FUNCTION_BLOCK FB_RateFromEPICS

(*
enum MPSBeamRates {
    MPSRateInvalid            =  0,
    MPSRate0Hz                =  1,
    /* Previously used 2 and 3 for single shot and burst */
    MPSRate1Hz                =  4,
    MPSRate10Hz               =  5,
    MPSRate30Hz               =  6,
    MPSRate60Hz               =  7,
    MPSRate120Hz              =  8,
    MPSRateUnknown            =  9,
    MPSRateSingleShot         = 10,
    MPSRateBurstMode          = 11,
    MPSRateBurstModeNotActive = 12,
    MPSNumberOfBeamRates      = 13,
    MPSRateBurstInvalid       = 14
}
*)

VAR_IN_OUT
    BP : ST_BeamParams;
    fbBYKIK_Rate : FB_LREALFromEPICS;
    FFO : FB_HardwareFFOutput;
END_VAR
VAR_OUTPUT
    xError : BOOL;
END_VAR
VAR


    eMPSRate : E_MPSBeamRates;

    ffRateReadBack : FB_FastFault := (
        i_DevName := 'Arbiter',
        i_Desc := 'Issue with rate readback from Accelerator. Gateway or EPICS connection. Must be fixed.',
        i_TypeCode := 16#203,
        i_xAutoReset:=True);
END_VAR
VAR CONSTANT
    cFailSafeRate : UDINT := 1000001;
END_VAR

fbBYKIK_Rate();

IF fbBYKIK_Rate.bValid THEN
    eMPSRate := LREAL_TO_UINT(fbBYKIK_Rate.fValue);
ELSE
    eMPSRate := E_MPSBeamRates.MPSRateInvalid;
END_IF

CASE eMPSRate OF
    MPSRateInvalid:
        BP.nRate := cFailSafeRate;
    MPSRate0Hz:
        BP.nRate := 0;
    MPSRate1Hz:
        BP.nRate := 1;
    MPSRate10Hz:
        BP.nRate := 10;
    MPSRate30Hz:
        BP.nRate := 30;
    MPSRate60Hz:
        BP.nRate := 60;
    MPSRate120Hz:
        BP.nRate := 120;
    MPSRateUnknown:
        BP.nRate := cFailSafeRate;

ELSE
    BP.nRate := cFailSafeRate;
END_CASE

ffRateReadback(i_xOK:=fbBYKIK_Rate.bValid, io_fbFFHWO:=FFO);

BP.xValid R= NOT fbBYKIK_Rate.bValid OR
            eMPSRate = MPSRateUnknown OR
            eMPSRate = MPSRateInvalid;

END_FUNCTION_BLOCK

(* stored: Version 1.1.0.1, ProductVersion 3.1.4022.18
   POU FB_RateFromEPICS: Id {1e21f3bc-80d5-47ca-8c4a-554964f1c13d}, SpecialFunc None *)
